{attribute 'qualified_only'}
{attribute 'strict'}
TYPE E_SHUTTER_HW_STATUS :
(
	UNKNOWN	:= 0,
	ERROR,
	CLOSED,
	OPEN
);
END_TYPE

(* stored: Version 1.1.0.1, ProductVersion 3.1.4022.16
   DUT E_SHUTTER_HW_STATUS: Id {114b996d-27ba-4ea5-8b3d-fdb43590f09c} *)
